(* PLC project Tc2_Standard.DELETE Demo, tc3-libraries-kb TwinCAT 3.1 *)
(* stored: creationDateTime 2026-05-10T08:00:00, modificationDateTime 2026-05-10T08:00:00 *)

PROGRAM P_Demo_DELETE
  VAR
    sResult : STRING;  (* DELETE 的返回值（监视） *)
    bRun : BOOL;  (* 触发一次 DELETE 调用 *)
  END_VAR

            // ============================================================
// Tc2_Standard.DELETE 演示程序（FUNCTION）
// ============================================================
// 场景：去掉中间 2 个字符
// 验证步骤：
//   1. 编译并登录目标
//   2. 强制 bRun := TRUE 一个周期
//   3. 观察 sResult = 'SUSI'
//   4. bRun 自动复位
// ============================================================

IF bRun THEN
    sResult := DELETE('SUXYSI',2,3);
    bRun := FALSE;
END_IF;

          
END_PROGRAM
